PROGRAM PRG_04_Turret
VAR

	lTurretCWLimit :LREAL;
	lTurretCCWLimit :LREAL;
	lTurretMedian: LREAL;
	lTurretEncoderValue: LREAL;
	R_TRIG_0: R_TRIG;
	R_TRIG_1: R_TRIG;
	R_TRIG_2: R_TRIG;
	R_TRIG_3: R_TRIG;
	R_TRIG_4: R_TRIG;
	R_TRIG_5: R_TRIG;
	RS_1: RS;
	R_TRIG_6: R_TRIG;
	R_TRIG_7: R_TRIG;
	SR_2: SR;
	R_TRIG_8: R_TRIG;
	R_TRIG_9: R_TRIG;
	RS_2: RS;
	R_TRIG_10: R_TRIG;
	R_TRIG_11: R_TRIG;
	SR_3: SR;
	RS_3: RS;
	R_TRIG_12: R_TRIG;
	R_TRIG_13: R_TRIG;
	R_TRIG_14: R_TRIG;
	R_TRIG_15: R_TRIG;
	bTurretRt: BOOL;
	bTurretLt: BOOL;

	dTurretEncoderValue: DINT;

	DINTmaxvalue: DINT;
	DINThalfvalue: DINT;
	dTurretCCWLimit: DINT;
	dTurretCWLimit: DINT;
	dTurretMedian: DINT;
END_VAR

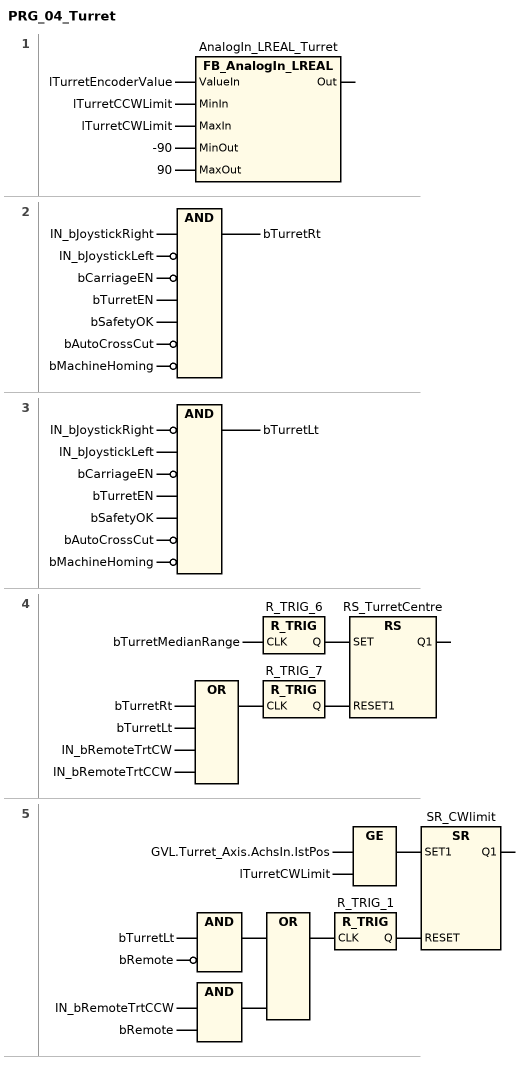
// NETWORK 1
AnalogIn_LREAL_Turret(
    ValueIn := lTurretEncoderValue,
    MinIn := lTurretCCWLimit,
    MaxIn := lTurretCWLimit,
    MinOut := -90,
    MaxOut := 90); // FB_AnalogIn_LREAL

// NETWORK 2
bTurretRt := IN_bJoystickRight AND NOT IN_bJoystickLeft AND NOT bCarriageEN AND bTurretEN AND bSafetyOK AND NOT bAutoCrossCut AND NOT bMachineHoming;

// NETWORK 3
bTurretLt := NOT IN_bJoystickRight AND IN_bJoystickLeft AND NOT bCarriageEN AND bTurretEN AND bSafetyOK AND NOT bAutoCrossCut AND NOT bMachineHoming;

// NETWORK 4
R_TRIG_6(CLK := bTurretMedianRange); // R_TRIG
R_TRIG_7(CLK := bTurretRt OR bTurretLt OR IN_bRemoteTrtCW OR IN_bRemoteTrtCCW); // R_TRIG
RS_TurretCentre(SET := R_TRIG_6.Q, RESET1 := R_TRIG_7.Q); // RS

// NETWORK 5
R_TRIG_1(CLK := bTurretLt AND NOT bRemote OR IN_bRemoteTrtCCW AND bRemote); // R_TRIG
SR_CWlimit(SET1 := GVL.Turret_Axis.AchsIn.IstPos >= lTurretCWLimit, RESET := R_TRIG_1.Q); // SR

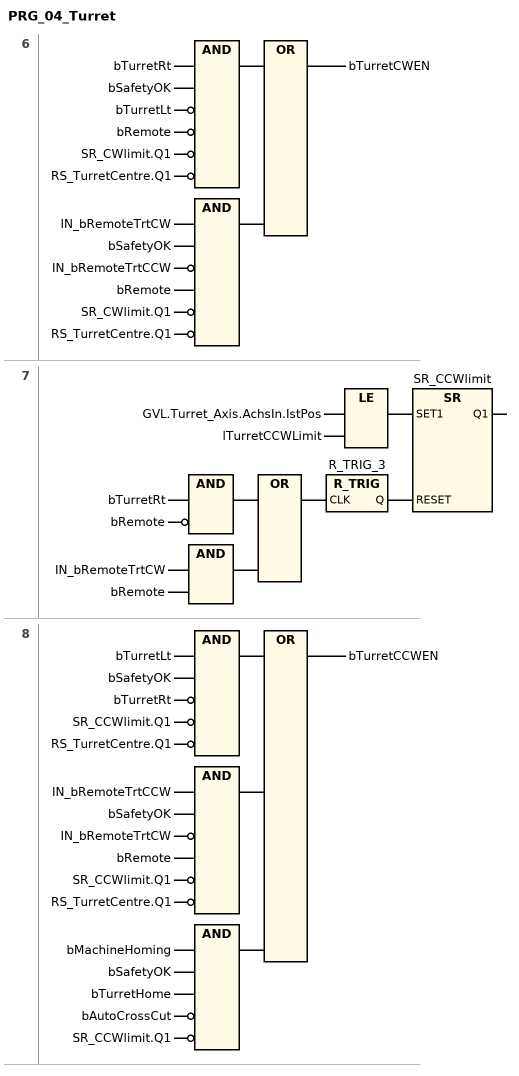
// NETWORK 6
bTurretCWEN := bTurretRt AND bSafetyOK AND NOT bTurretLt AND NOT bRemote AND NOT SR_CWlimit.Q1 AND NOT RS_TurretCentre.Q1 OR IN_bRemoteTrtCW AND bSafetyOK AND NOT IN_bRemoteTrtCCW AND bRemote AND NOT SR_CWlimit.Q1 AND NOT RS_TurretCentre.Q1;

// NETWORK 7
R_TRIG_3(CLK := bTurretRt AND NOT bRemote OR IN_bRemoteTrtCW AND bRemote); // R_TRIG
SR_CCWlimit(SET1 := GVL.Turret_Axis.AchsIn.IstPos <= lTurretCCWLimit, RESET := R_TRIG_3.Q); // SR

// NETWORK 8
bTurretCCWEN := bTurretLt AND bSafetyOK AND NOT bTurretRt AND NOT SR_CCWlimit.Q1 AND NOT RS_TurretCentre.Q1 OR IN_bRemoteTrtCCW AND bSafetyOK AND NOT IN_bRemoteTrtCW AND bRemote AND NOT SR_CCWlimit.Q1 AND NOT RS_TurretCentre.Q1 OR bMachineHoming AND bSafetyOK AND bTurretHome AND NOT bAutoCrossCut AND NOT SR_CCWlimit.Q1;

ACTION ACT_04_1_Turret:
lTurretMedian := 1295.531998;	// square the CROSSCUT subassy, not the saw blade!!!
lTurretCWLimit := lTurretMedian + 319.7995;
lTurretCCWLimit := lTurretMedian - 319.7995;

(* Turret encoder rollover *)
IF lTurretEncoderValue < lTurretCCWLimit THEN
	lTurretEncoderValue := lTurretCCWLimit ;
ELSIF lTurretEncoderValue > lTurretCWLimit THEN
	lTurretEncoderValue := lTurretCWLimit ;
ELSE 
	lTurretEncoderValue := GVL.Turret_Axis.AchsIn.IstPos ;
END_IF

(* Turret slow downs approaching 90°, -90° end limits and 0° *)	
IF  (AnalogIn_LREAL_Turret.Out.rScaled >= 88 AND (bTurretRt OR (IN_bRemoteTrtCW AND bRemote) OR (bTurretHome AND bMachineHoming))) OR
	(AnalogIn_LREAL_Turret.Out.rScaled <= -88 AND (bTurretLt OR (IN_bRemoteTrtCCW AND bRemote) OR (bTurretHome AND bMachineHoming))) OR
	(AnalogIn_LREAL_Turret.Out.rScaled >= -2 AND AnalogIn_LREAL_Turret.Out.rScaled < 0 AND (bTurretRt OR (IN_bRemoteTrtCW AND bRemote))) OR
	(AnalogIn_LREAL_Turret.Out.rScaled <= 2 AND AnalogIn_LREAL_Turret.Out.rScaled > 0 AND (bTurretLt OR (IN_bRemoteTrtCCW AND bRemote)))
THEN
	bTurretJogFast := FALSE ;
ELSE
	bTurretJogFast := TRUE ;
END_IF

(* Trigger stop turret at ~0° *)
IF GVL.Turret_Axis.AchsIn.IstPos > lTurretMedian - 0.01 AND
	GVL.Turret_Axis.AchsIn.IstPos < lTurretMedian + 0.01
THEN
	bTurretMedianRange := TRUE ;
ELSE bTurretMedianRange := FALSE ;
END_IF

(* Turret 45° range *)
IF AnalogIn_LREAL_Turret.Out.rScaled < 47 AND AnalogIn_LREAL_Turret.Out.rScaled > -47 THEN
	bTurret045Range := TRUE ;
ELSE bTurret045Range := FALSE ;
END_IF
END_ACTION

END_PROGRAM

(* stored: Version 1.1.0.1, ProductVersion 3.1.4024.15
   POU PRG_04_Turret: Id {68211daf-2798-43fd-94be-d04d278eca53}, SpecialFunc None
   Action ACT_04_1_Turret: Id {c42e3bb7-9e23-4d2c-b2d4-7fae912b0bb1} *)
